# EPICS substitutions: SRS_PS300Sup/devSRS_PS365.substitutions
##########################################################################
# Copyright (c) 2012 Lawrence Berkeley National Laboratory, Accelerator
# Technology Group, Engineering Division
# This code is distributed subject to a Software License Agreement found
# in file LICENSE that is included with this distribution.
##########################################################################

file devSRS_PS3xx.template
{
  { P="\$(P)", R="\$(R)", PORT="\$(PORT)", A="\$(A)",
  VMIN="100", VMAX="10000", IMIN="0", IMAX="1e-3" }
}
